{attribute 'qualified_only'}
VAR_GLOBAL
	GC1 : ST_GC_Ctrl;
END_VAR

(* stored: Version 1.1.0.1, ProductVersion 3.1.4026.18
   GVL GVL_CSharp: Id {2ccf78e0-eb9f-46e8-912a-067d5425c8dd} *)
